Staubli VAL3: printBool.pgx

public program printBool(bool& x_bInput[])
  local num l_nElement
  local num l_nLength
begin

  l_nLength = size(x_bInput)

  for l_nElement = 0 to l_nLength-1
    ? x_bInput[l_nElement]
  endFor

end
